// TIA Portal V18 export
TYPE "UDT_Store_Season"
// stored: IsFailsafeCompliant false
   STRUCT
      cSeasonModeSelection : Byte;   // 0 = Summer 1 = Winter 2 = Midseason, 3=Auro
      cActual : Byte;   // 0 = Summer 1 = Winter 2 = Midseason
      cTarget : Byte;
      cReserve : Byte;
      rOATtoWinter : Real := 10.0;
      rOATtoSummer : Real := 12.0;
   END_STRUCT;
END_TYPE
